FUNCTION_BLOCK Sensor_HMI (* Service Interface Function Block Type *)
  (* Standard: 61499-2 *)
  (* Version 0.0, 9/14/2008, Horst Mayer, nxtControl GmbH, template *)
  PACKAGE Main;
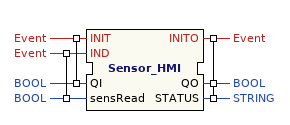
  EVENT_INPUT
    INIT WITH QI;
    IND WITH sensRead;
  END_EVENT
  EVENT_OUTPUT
    INITO WITH QO, STATUS;
  END_EVENT
  VAR_INPUT
    QI : BOOL;
    sensRead : BOOL;
  END_VAR
  VAR_OUTPUT
    QO : BOOL; (* Event Output Qualifier *)
    STATUS : STRING; (* Service Status *)
  END_VAR
END_FUNCTION_BLOCK
